FUNCTION_BLOCK TestSuite EXTENDS FB_TestSuite

END_FUNCTION_BLOCK

(* stored: Version 1.1.0.1, ProductVersion 3.1.4024.6
   POU TestSuite: Id {a7e22833-6c27-466d-9ad3-520ef4a39cff}, SpecialFunc None *)
